TYPE ST_ValveFeedback_1 :
STRUCT
	sName : STRING(8);
END_STRUCT
END_TYPE

(* stored: Version 1.1.0.1, ProductVersion 3.1.4024.12
   DUT ST_ValveFeedback_1: Id {67a2f32f-6a92-48ff-b744-64efa2fa04ee} *)
